{attribute 'qualified_only'}
{attribute 'strict'}
TYPE E_RecoveryState :
(

	Idle 						:= 0,
	Metering_Solvent1 			:= 1,
	Recirculate_Solvent1 		:= 2,
	Solvent_Soak 				:= 3,
	Cleaning_Lines_S1 			:= 4,
	Metering_Solvent2 			:= 5,
	AgitateTime1				:= 6,
	Mix_Solvent1_2 				:= 7,
	Cleaning_Lines_S1_S2 		:= 8,
	AgitateTime2				:= 9,
	Prime_Needles 				:= 10,
	Fill_Vials_Row_1 			:= 11,
	Fill_Vials_Row_2 			:= 12,
	Fill_Vials_Row_3 			:= 13,
	Fill_Vials_Row_4 			:= 14,
	Waste_Remaining_Solvent 	:= 15,
	Completed 					:= 16,
	Error						:= 17

);
END_TYPE

(* stored: Version 1.1.0.1, ProductVersion 3.1.4024.15
   DUT E_RecoveryState: Id {0cfef865-1384-4e4a-be3f-5c996ab7a8f8} *)
